// TIA Portal project "MYJZXT_PLC" (V15.1)
// 煤油加注系统(新)

(* hardware
DEVICE "S7-1200 station_1"  S7-1200 Station
   slot 0: "Rack_0"  S7-1200 Rack  Rack  V1.0
   slot 1: "PLC_1"  CPU 1215C DC/DC/Rly  6ES7 215-1HG40-0XB0  V4.2
   slot 2: "AI 8x13BIT_1"  6ES7 231-4HF32-0XB0  V2.0
   slot 3: "CB 1241 (RS485)"  CB 1241 (RS485)  6ES7 241-1CH30-1XB0  V1.0
   slot 3: "AI 8x13BIT_2"  6ES7 231-4HF32-0XB0  V2.0
   slot 4: "DI 8/DQ 8x24VDC_1"  6ES7 223-1BH32-0XB0  V2.0
*)

// ===== PLC "PLC_1"  CPU 1215C DC/DC/Rly =====

VAR_GLOBAL   // PLC tag table "默认变量表"
   "Pc0_int" AT %IW96 : Int;
   "中间变量1" AT %MD10 : Real;
   "Pc0_real" AT %MD14 : Real;
   "Pc1_int" AT %IW98 : Int;
   "Pc1_real" AT %MD18 : Real;
   "Pc2_int" AT %IW100 : Int;
   "Pc2_real" AT %MD22 : Real;
   "Pc3_int" AT %IW102 : Int;
   "Pc3_real" AT %MD26 : Real;
   "Pc4_int" AT %IW104 : Int;
   "Pc4_real" AT %MD30 : Real;
   "Pc5_int" AT %IW106 : Int;
   "Pc5_real" AT %MD34 : Real;
   "YW01_real" AT %MD38 : Real;
   "YW02_real" AT %MD42 : Real;
   "YW01_int" AT %IW112 : Int;
   "YW02_int" AT %IW114 : Int;
   "YW03_int" AT %IW116 : Int;
   "PD01" AT %IW118 : Int;
   "PD02" AT %IW120 : Int;
   "PD01_real" AT %MD50 : Real;
   "PD02_real" AT %MD54 : Real;
   "急停" AT %I0.0 : Bool;
   "变频器" AT %QW64 : Int;
   "转注泵" AT %Q0.0 : Bool;
   "加注泵" AT %Q0.1 : Bool;
   "真空泵" AT %Q0.2 : Bool;
   "DC01" AT %Q16.0 : Bool;
   "DC02" AT %Q16.1 : Bool;
   "DC03" AT %Q16.2 : Bool;
   "DC04" AT %Q16.3 : Bool;
   "DC05" AT %Q16.4 : Bool;
   "DC06" AT %Q16.5 : Bool;
   "DC07" AT %Q16.6 : Bool;
   "DC08" AT %Q16.7 : Bool;
   "变频设置" AT %MW58 : Int;
   "转注总流量" AT %MD60 : Real;
   "加注总流量" AT %MD64 : Real;
   "转注设定量" AT %MD68 : Real;
   "加注设定量" AT %MD72 : Real;
   "回排设定量" AT %MD76 : Real;
   "真空度" AT %MD6 : Real;
   "~真空加注完成" AT %M100.0 : Bool;
   "抽真空自检成功" AT %M100.1 : Bool;
   "真空加注真空自检成功" AT %M100.2 : Bool;
   "真空加注完成" AT %M100.3 : Bool;
   "回排结束标志" AT %M100.4 : Bool;
   "清洁结束" AT %M100.5 : Bool;
   "YW03_real" AT %MD46 : Real;
   "液路自检完成" AT %M100.6 : Bool;
   "转注完成" AT %M100.7 : Bool;
   "pc0" AT %MW80 : Int;
   "pc1" AT %MW82 : Int;
   "pc2" AT %MW84 : Int;
   "pc3" AT %MW86 : Int;
   "pc4" AT %MW88 : Int;
   "pc5" AT %MW90 : Int;
   "yw01" AT %MW92 : Int;
   "yw02" AT %MW94 : Int;
   "yw03" AT %MW96 : Int;
   "pd1" AT %MW98 : Int;
   "pd2" AT %MW110 : Int;
   "中间变量2" AT %MD106 : Real;
   "pip_tmp1" AT %M5.0 : Bool;
   "pip_tmp2" AT %M5.1 : Bool;
   "中间变量3" AT %MD112 : Real;
   "转/回总流量" AT %MW116 : Word;
   "加总流量" AT %MW118 : Int;
   "流量设定中间变量" AT %MW122 : Word;
   "System_Byte" AT %MB1 : Byte;
   "FirstScan" AT %M1.0 : Bool;
   "DiagStatusUpdate" AT %M1.1 : Bool;
   "AlwaysTRUE" AT %M1.2 : Bool;
   "AlwaysFALSE" AT %M1.3 : Bool;
END_VAR

VAR_GLOBAL   // PLC tag table "control"
   "current_index" AT %MB120 : Byte;   // 当前流程
   "startORstop" AT %MB124 : Byte;   // 流程开始/结束状态
   "setTime" AT %MD125 : Time;
   "current_step" AT %MB121 : Byte;
   "setZKD" AT %MW130 : Int;
   "setZKD_1" AT %MW132 : Int;
   "ZKD_keep" AT %MD134 : Real;
   "转注_set" AT %MW138 : UInt;
END_VAR

DATA_BLOCK "zhuanzhu_flow"   // DB7
{ S7_Optimized_Access := 'TRUE' }
VERSION : 0.1
// stored: InstanceOfName Flowcalc
"Flowcalc"
BEGIN
END_DATA_BLOCK

DATA_BLOCK "jiazhu_flow"   // DB8
{ S7_Optimized_Access := 'TRUE' }
VERSION : 0.1
// stored: InstanceOfName Flowcalc
"Flowcalc"
BEGIN
END_DATA_BLOCK

DATA_BLOCK "tcp_DB"   // DB9
{ S7_Optimized_Access := 'FALSE' }
VERSION : 0.1
   VAR
      ToClientArray : Array[0..50] of Byte;
      FromClientArray : Array[0..20] of Byte;
   END_VAR
BEGIN
END_DATA_BLOCK

DATA_BLOCK "tcp_status"   // DB13
{ S7_Optimized_Access := 'TRUE' }
VERSION : 0.1
   VAR
      TRCV_DONE : Bool;
      TRCV_BUSY : Bool;
      TRCV_ERROR : Bool;
      TRCV_STATUS : Word;
      TRCV_LEGNTH : UDInt;
      TSEND_DONE : Bool;
      TSEND_STATUS : Word;
      TSEND_BUSY : Bool;
      TSEND_REQ : Bool := true;
      TSEND_ERROR : Bool;
   END_VAR
BEGIN
END_DATA_BLOCK

DATA_BLOCK "485_db"   // DB30
{ S7_Optimized_Access := 'TRUE' }
VERSION : 0.1
   VAR
      "485_data" : Array[0..7] of Byte;
   END_VAR
BEGIN
END_DATA_BLOCK

// folder: System blocks/Program resources

DATA_BLOCK "timer_ylzj"   // DB1
{ S7_Optimized_Access := 'TRUE' }
AUTHOR : Simatic
FAMILY : IEC
NAME : IEC_TMR
VERSION : 1.0
// stored: InstanceOfName IEC_TIMER
"IEC_TIMER"
BEGIN
END_DATA_BLOCK

DATA_BLOCK "timer_czkzj"   // DB2
{ S7_Optimized_Access := 'TRUE' }
AUTHOR : Simatic
FAMILY : IEC
NAME : IEC_TMR
VERSION : 1.0
// stored: InstanceOfName IEC_TIMER
"IEC_TIMER"
BEGIN
END_DATA_BLOCK

DATA_BLOCK "timer_ZKD_keep"   // DB3
{ S7_Optimized_Access := 'TRUE' }
AUTHOR : Simatic
FAMILY : IEC
NAME : IEC_TMR
VERSION : 1.0
// stored: InstanceOfName IEC_TIMER
"IEC_TIMER"
BEGIN
END_DATA_BLOCK

DATA_BLOCK "timer_cqsj"   // DB4
{ S7_Optimized_Access := 'TRUE' }
AUTHOR : Simatic
FAMILY : IEC
NAME : IEC_TMR
VERSION : 1.0
// stored: InstanceOfName IEC_TIMER
"IEC_TIMER"
BEGIN
END_DATA_BLOCK

DATA_BLOCK "timer_cz"   // DB5
{ S7_Optimized_Access := 'TRUE' }
AUTHOR : Simatic
FAMILY : IEC
NAME : IEC_TMR
VERSION : 1.0
// stored: InstanceOfName IEC_TIMER
"IEC_TIMER"
BEGIN
END_DATA_BLOCK

DATA_BLOCK "timer_keeper"   // DB6
{ S7_Optimized_Access := 'TRUE' }
AUTHOR : Simatic
FAMILY : IEC
NAME : IEC_TMR
VERSION : 1.0
// stored: InstanceOfName IEC_TIMER
"IEC_TIMER"
BEGIN
END_DATA_BLOCK

DATA_BLOCK "PLC_1_Receive_DB"   // DB12
{ S7_Optimized_Access := 'TRUE' }
AUTHOR : SIMATIC
FAMILY : MC7Plus
NAME : TC_IP_v4
VERSION : 1.0
// stored: InstanceOfName TCON_IP_v4
"TCON_IP_v4"
BEGIN
   ID := 1;
   InterfaceId := 64;
   LocalPort := 2000;
   RemoteAddress.ADDR[1] := 192;
   RemoteAddress.ADDR[2] := 168;
   RemoteAddress.ADDR[3] := 2;
   RemoteAddress.ADDR[4] := 3;
END_DATA_BLOCK

DATA_BLOCK "timer_delay2"   // DB16
{ S7_Optimized_Access := 'TRUE' }
AUTHOR : Simatic
FAMILY : IEC
NAME : IEC_TMR
VERSION : 1.0
// stored: InstanceOfName IEC_TIMER
"IEC_TIMER"
BEGIN
END_DATA_BLOCK

DATA_BLOCK "IEC_Timer_0_DB_1"   // DB17
{ S7_Optimized_Access := 'TRUE' }
AUTHOR : Simatic
FAMILY : IEC
NAME : IEC_TMR
VERSION : 1.0
// stored: InstanceOfName IEC_TIMER
"IEC_TIMER"
BEGIN
END_DATA_BLOCK

DATA_BLOCK "send_delay"   // DB26
{ S7_Optimized_Access := 'TRUE' }
AUTHOR : Simatic
FAMILY : IEC
NAME : IEC_TMR
VERSION : 1.0
// stored: InstanceOfName IEC_TIMER
"IEC_TIMER"
BEGIN
END_DATA_BLOCK

DATA_BLOCK "send_delay1"   // DB27
{ S7_Optimized_Access := 'TRUE' }
AUTHOR : Simatic
FAMILY : IEC
NAME : IEC_TMR
VERSION : 1.0
// stored: InstanceOfName IEC_TIMER
"IEC_TIMER"
BEGIN
END_DATA_BLOCK

// folder: (top level)

FUNCTION_BLOCK "Flowcalc"   // FB1, SCL
{ S7_Optimized_Access := 'TRUE' }
VERSION : 0.1
   VAR_INPUT
      flow : Real;
      Enable : Bool;
   END_VAR
   VAR_OUTPUT
      sum : Real;
   END_VAR
   VAR
      data : Real;
   END_VAR
BEGIN
   IF #Enable = FALSE THEN
       #data := 0.0;
       ;
   ELSE
       IF #flow > 1.0 THEN
           #data := #data + #flow / 60 * 0.1;
           #sum := #data;
       ELSE
           #sum := #data;
       END_IF;
       // Statement section IF
       ;
   END_IF;
END_FUNCTION_BLOCK

FUNCTION "模拟量采集" : Void   // FC1, LAD
{ S7_Optimized_Access := 'TRUE' }
VERSION : 0.1
BEGIN

REGION Network 1
   // 压力传感器0
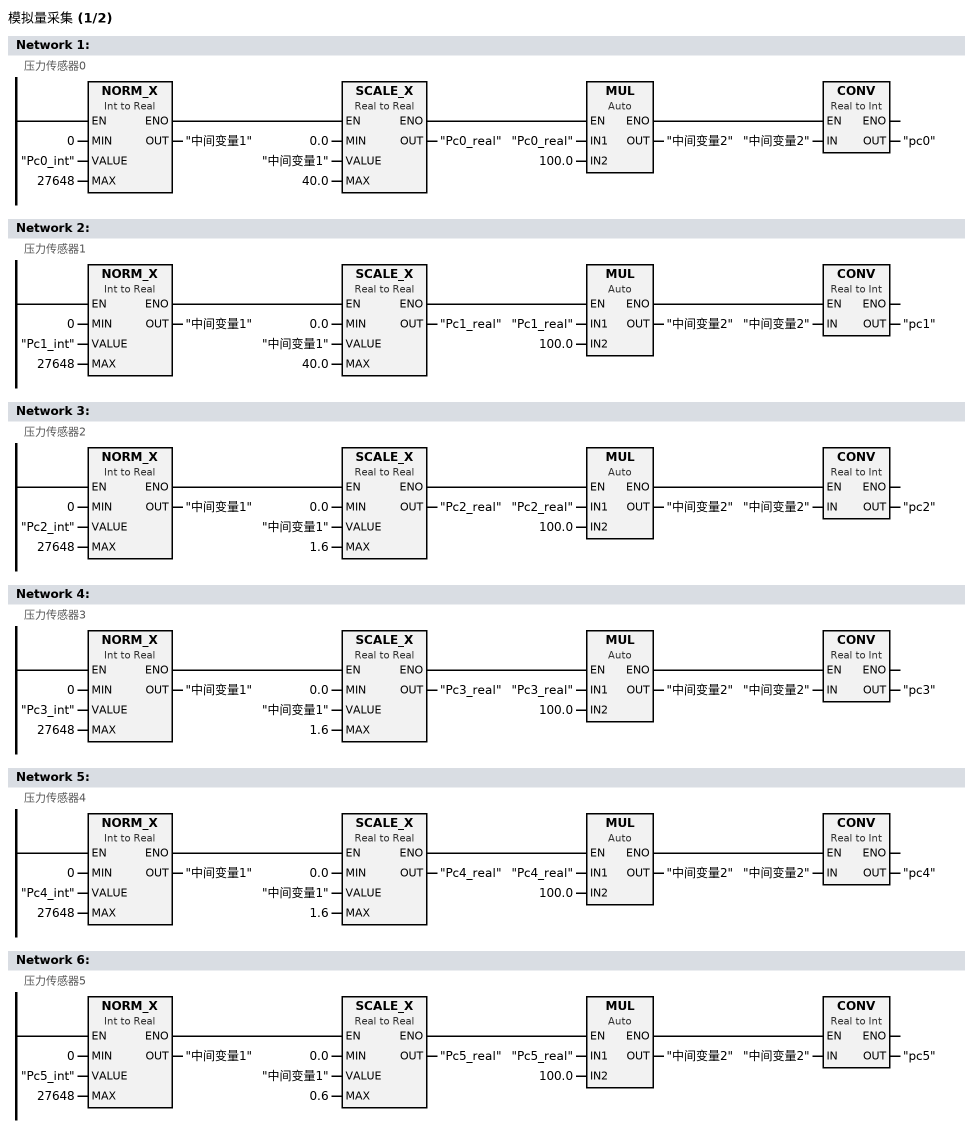
   RUNG wire#powerrail
      { S7_Templates := "[SrcType := Int, DestType := Real]"; S7_GenerateENO := "TRUE" } Normalize(min := 0, value := "Pc0_int", max := 27648, out => "中间变量1")
      { S7_Templates := "[SrcType := Real, DestType := Real]"; S7_GenerateENO := "TRUE" } Scale(min := 0.0, value := "中间变量1", max := 40.0, out => "Pc0_real")
      { S7_GenerateENO := "TRUE" } Mul(in1 := "Pc0_real", in2 := 100.0, out => "中间变量2")
      { S7_Templates := "[SrcType := Real, DestType := Int]"; S7_GenerateENO := "TRUE" } Convert(in := "中间变量2", out => "pc0")
   END_RUNG
   // the same network as SCL:
   // ENO of a box is taken as its EN; it also drops when the box reports an error
   "中间变量1" := NORM_X(MIN := 0, VALUE := "Pc0_int", MAX := 27648);
   "Pc0_real" := SCALE_X(MIN := 0.0, VALUE := "中间变量1", MAX := 40.0);
   "中间变量2" := "Pc0_real" * 100.0;
   "pc0" := REAL_TO_INT("中间变量2");
END_REGION

REGION Network 2
   // 压力传感器1
   RUNG wire#powerrail
      { S7_Templates := "[SrcType := Int, DestType := Real]"; S7_GenerateENO := "TRUE" } Normalize(min := 0, value := "Pc1_int", max := 27648, out => "中间变量1")
      { S7_Templates := "[SrcType := Real, DestType := Real]"; S7_GenerateENO := "TRUE" } Scale(min := 0.0, value := "中间变量1", max := 40.0, out => "Pc1_real")
      { S7_GenerateENO := "TRUE" } Mul(in1 := "Pc1_real", in2 := 100.0, out => "中间变量2")
      { S7_Templates := "[SrcType := Real, DestType := Int]"; S7_GenerateENO := "TRUE" } Convert(in := "中间变量2", out => "pc1")
   END_RUNG
   // the same network as SCL:
   // ENO of a box is taken as its EN; it also drops when the box reports an error
   "中间变量1" := NORM_X(MIN := 0, VALUE := "Pc1_int", MAX := 27648);
   "Pc1_real" := SCALE_X(MIN := 0.0, VALUE := "中间变量1", MAX := 40.0);
   "中间变量2" := "Pc1_real" * 100.0;
   "pc1" := REAL_TO_INT("中间变量2");
END_REGION

REGION Network 3
   // 压力传感器2
   RUNG wire#powerrail
      { S7_Templates := "[SrcType := Int, DestType := Real]"; S7_GenerateENO := "TRUE" } Normalize(min := 0, value := "Pc2_int", max := 27648, out => "中间变量1")
      { S7_Templates := "[SrcType := Real, DestType := Real]"; S7_GenerateENO := "TRUE" } Scale(min := 0.0, value := "中间变量1", max := 1.6, out => "Pc2_real")
      { S7_GenerateENO := "TRUE" } Mul(in1 := "Pc2_real", in2 := 100.0, out => "中间变量2")
      { S7_Templates := "[SrcType := Real, DestType := Int]"; S7_GenerateENO := "TRUE" } Convert(in := "中间变量2", out => "pc2")
   END_RUNG
   // the same network as SCL:
   // ENO of a box is taken as its EN; it also drops when the box reports an error
   "中间变量1" := NORM_X(MIN := 0, VALUE := "Pc2_int", MAX := 27648);
   "Pc2_real" := SCALE_X(MIN := 0.0, VALUE := "中间变量1", MAX := 1.6);
   "中间变量2" := "Pc2_real" * 100.0;
   "pc2" := REAL_TO_INT("中间变量2");
END_REGION

REGION Network 4
   // 压力传感器3
   RUNG wire#powerrail
      { S7_Templates := "[SrcType := Int, DestType := Real]"; S7_GenerateENO := "TRUE" } Normalize(min := 0, value := "Pc3_int", max := 27648, out => "中间变量1")
      { S7_Templates := "[SrcType := Real, DestType := Real]"; S7_GenerateENO := "TRUE" } Scale(min := 0.0, value := "中间变量1", max := 1.6, out => "Pc3_real")
      { S7_GenerateENO := "TRUE" } Mul(in1 := "Pc3_real", in2 := 100.0, out => "中间变量2")
      { S7_Templates := "[SrcType := Real, DestType := Int]"; S7_GenerateENO := "TRUE" } Convert(in := "中间变量2", out => "pc3")
   END_RUNG
   // the same network as SCL:
   // ENO of a box is taken as its EN; it also drops when the box reports an error
   "中间变量1" := NORM_X(MIN := 0, VALUE := "Pc3_int", MAX := 27648);
   "Pc3_real" := SCALE_X(MIN := 0.0, VALUE := "中间变量1", MAX := 1.6);
   "中间变量2" := "Pc3_real" * 100.0;
   "pc3" := REAL_TO_INT("中间变量2");
END_REGION

REGION Network 5
   // 压力传感器4
   RUNG wire#powerrail
      { S7_Templates := "[SrcType := Int, DestType := Real]"; S7_GenerateENO := "TRUE" } Normalize(min := 0, value := "Pc4_int", max := 27648, out => "中间变量1")
      { S7_Templates := "[SrcType := Real, DestType := Real]"; S7_GenerateENO := "TRUE" } Scale(min := 0.0, value := "中间变量1", max := 1.6, out => "Pc4_real")
      { S7_GenerateENO := "TRUE" } Mul(in1 := "Pc4_real", in2 := 100.0, out => "中间变量2")
      { S7_Templates := "[SrcType := Real, DestType := Int]"; S7_GenerateENO := "TRUE" } Convert(in := "中间变量2", out => "pc4")
   END_RUNG
   // the same network as SCL:
   // ENO of a box is taken as its EN; it also drops when the box reports an error
   "中间变量1" := NORM_X(MIN := 0, VALUE := "Pc4_int", MAX := 27648);
   "Pc4_real" := SCALE_X(MIN := 0.0, VALUE := "中间变量1", MAX := 1.6);
   "中间变量2" := "Pc4_real" * 100.0;
   "pc4" := REAL_TO_INT("中间变量2");
END_REGION

REGION Network 6
   // 压力传感器5
   RUNG wire#powerrail
      { S7_Templates := "[SrcType := Int, DestType := Real]"; S7_GenerateENO := "TRUE" } Normalize(min := 0, value := "Pc5_int", max := 27648, out => "中间变量1")
      { S7_Templates := "[SrcType := Real, DestType := Real]"; S7_GenerateENO := "TRUE" } Scale(min := 0.0, value := "中间变量1", max := 0.6, out => "Pc5_real")
      { S7_GenerateENO := "TRUE" } Mul(in1 := "Pc5_real", in2 := 100.0, out => "中间变量2")
      { S7_Templates := "[SrcType := Real, DestType := Int]"; S7_GenerateENO := "TRUE" } Convert(in := "中间变量2", out => "pc5")
   END_RUNG
   // the same network as SCL:
   // ENO of a box is taken as its EN; it also drops when the box reports an error
   "中间变量1" := NORM_X(MIN := 0, VALUE := "Pc5_int", MAX := 27648);
   "Pc5_real" := SCALE_X(MIN := 0.0, VALUE := "中间变量1", MAX := 0.6);
   "中间变量2" := "Pc5_real" * 100.0;
   "pc5" := REAL_TO_INT("中间变量2");
END_REGION

REGION Network 7
   // 液位计yw01
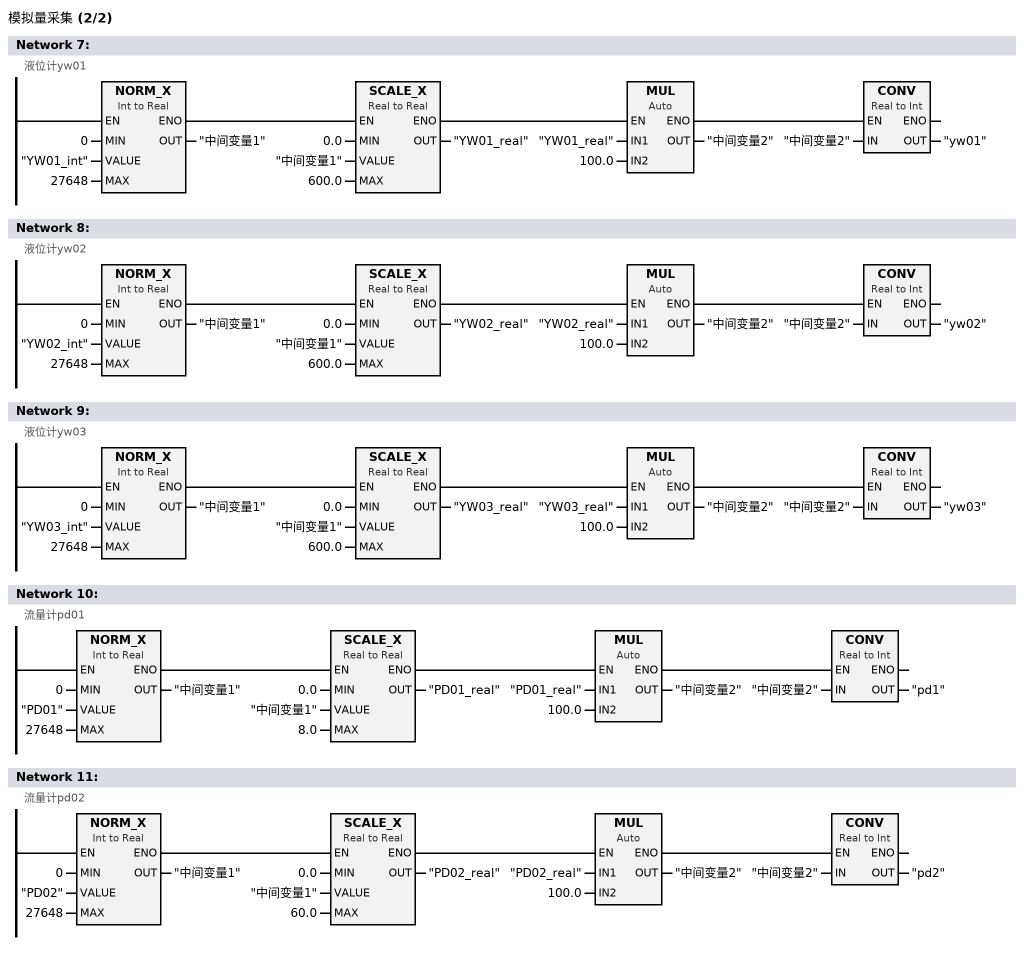
   RUNG wire#powerrail
      { S7_Templates := "[SrcType := Int, DestType := Real]"; S7_GenerateENO := "TRUE" } Normalize(min := 0, value := "YW01_int", max := 27648, out => "中间变量1")
      { S7_Templates := "[SrcType := Real, DestType := Real]"; S7_GenerateENO := "TRUE" } Scale(min := 0.0, value := "中间变量1", max := 600.0, out => "YW01_real")
      { S7_GenerateENO := "TRUE" } Mul(in1 := "YW01_real", in2 := 100.0, out => "中间变量2")
      { S7_Templates := "[SrcType := Real, DestType := Int]"; S7_GenerateENO := "TRUE" } Convert(in := "中间变量2", out => "yw01")
   END_RUNG
   // the same network as SCL:
   // ENO of a box is taken as its EN; it also drops when the box reports an error
   "中间变量1" := NORM_X(MIN := 0, VALUE := "YW01_int", MAX := 27648);
   "YW01_real" := SCALE_X(MIN := 0.0, VALUE := "中间变量1", MAX := 600.0);
   "中间变量2" := "YW01_real" * 100.0;
   "yw01" := REAL_TO_INT("中间变量2");
END_REGION

REGION Network 8
   // 液位计yw02
   RUNG wire#powerrail
      { S7_Templates := "[SrcType := Int, DestType := Real]"; S7_GenerateENO := "TRUE" } Normalize(min := 0, value := "YW02_int", max := 27648, out => "中间变量1")
      { S7_Templates := "[SrcType := Real, DestType := Real]"; S7_GenerateENO := "TRUE" } Scale(min := 0.0, value := "中间变量1", max := 600.0, out => "YW02_real")
      { S7_GenerateENO := "TRUE" } Mul(in1 := "YW02_real", in2 := 100.0, out => "中间变量2")
      { S7_Templates := "[SrcType := Real, DestType := Int]"; S7_GenerateENO := "TRUE" } Convert(in := "中间变量2", out => "yw02")
   END_RUNG
   // the same network as SCL:
   // ENO of a box is taken as its EN; it also drops when the box reports an error
   "中间变量1" := NORM_X(MIN := 0, VALUE := "YW02_int", MAX := 27648);
   "YW02_real" := SCALE_X(MIN := 0.0, VALUE := "中间变量1", MAX := 600.0);
   "中间变量2" := "YW02_real" * 100.0;
   "yw02" := REAL_TO_INT("中间变量2");
END_REGION

REGION Network 9
   // 液位计yw03
   RUNG wire#powerrail
      { S7_Templates := "[SrcType := Int, DestType := Real]"; S7_GenerateENO := "TRUE" } Normalize(min := 0, value := "YW03_int", max := 27648, out => "中间变量1")
      { S7_Templates := "[SrcType := Real, DestType := Real]"; S7_GenerateENO := "TRUE" } Scale(min := 0.0, value := "中间变量1", max := 600.0, out => "YW03_real")
      { S7_GenerateENO := "TRUE" } Mul(in1 := "YW03_real", in2 := 100.0, out => "中间变量2")
      { S7_Templates := "[SrcType := Real, DestType := Int]"; S7_GenerateENO := "TRUE" } Convert(in := "中间变量2", out => "yw03")
   END_RUNG
   // the same network as SCL:
   // ENO of a box is taken as its EN; it also drops when the box reports an error
   "中间变量1" := NORM_X(MIN := 0, VALUE := "YW03_int", MAX := 27648);
   "YW03_real" := SCALE_X(MIN := 0.0, VALUE := "中间变量1", MAX := 600.0);
   "中间变量2" := "YW03_real" * 100.0;
   "yw03" := REAL_TO_INT("中间变量2");
END_REGION

REGION Network 10
   // 流量计pd01
   RUNG wire#powerrail
      { S7_Templates := "[SrcType := Int, DestType := Real]"; S7_GenerateENO := "TRUE" } Normalize(min := 0, value := "PD01", max := 27648, out => "中间变量1")
      { S7_Templates := "[SrcType := Real, DestType := Real]"; S7_GenerateENO := "TRUE" } Scale(min := 0.0, value := "中间变量1", max := 8.0, out => "PD01_real")
      { S7_GenerateENO := "TRUE" } Mul(in1 := "PD01_real", in2 := 100.0, out => "中间变量2")
      { S7_Templates := "[SrcType := Real, DestType := Int]"; S7_GenerateENO := "TRUE" } Convert(in := "中间变量2", out => "pd1")
   END_RUNG
   // the same network as SCL:
   // ENO of a box is taken as its EN; it also drops when the box reports an error
   "中间变量1" := NORM_X(MIN := 0, VALUE := "PD01", MAX := 27648);
   "PD01_real" := SCALE_X(MIN := 0.0, VALUE := "中间变量1", MAX := 8.0);
   "中间变量2" := "PD01_real" * 100.0;
   "pd1" := REAL_TO_INT("中间变量2");
END_REGION

REGION Network 11
   // 流量计pd02
   RUNG wire#powerrail
      { S7_Templates := "[SrcType := Int, DestType := Real]"; S7_GenerateENO := "TRUE" } Normalize(min := 0, value := "PD02", max := 27648, out => "中间变量1")
      { S7_Templates := "[SrcType := Real, DestType := Real]"; S7_GenerateENO := "TRUE" } Scale(min := 0.0, value := "中间变量1", max := 60.0, out => "PD02_real")
      { S7_GenerateENO := "TRUE" } Mul(in1 := "PD02_real", in2 := 100.0, out => "中间变量2")
      { S7_Templates := "[SrcType := Real, DestType := Int]"; S7_GenerateENO := "TRUE" } Convert(in := "中间变量2", out => "pd2")
   END_RUNG
   // the same network as SCL:
   // ENO of a box is taken as its EN; it also drops when the box reports an error
   "中间变量1" := NORM_X(MIN := 0, VALUE := "PD02", MAX := 27648);
   "PD02_real" := SCALE_X(MIN := 0.0, VALUE := "中间变量1", MAX := 60.0);
   "中间变量2" := "PD02_real" * 100.0;
   "pd2" := REAL_TO_INT("中间变量2");
END_REGION
END_FUNCTION

FUNCTION "气路自检" : Void   // FC2, LAD
{ S7_Optimized_Access := 'TRUE' }
VERSION : 0.1
BEGIN

REGION Network 1: /气路自检为手动控制,当前无设置流程
END_REGION
END_FUNCTION

FUNCTION "液路自检" : Void   // FC3, LAD
{ S7_Optimized_Access := 'TRUE' }
VERSION : 0.1
   VAR_TEMP   // added for the SCL form of the ladder/FBD networks
      _w1 : Bool;
   END_VAR
BEGIN

REGION Network 1
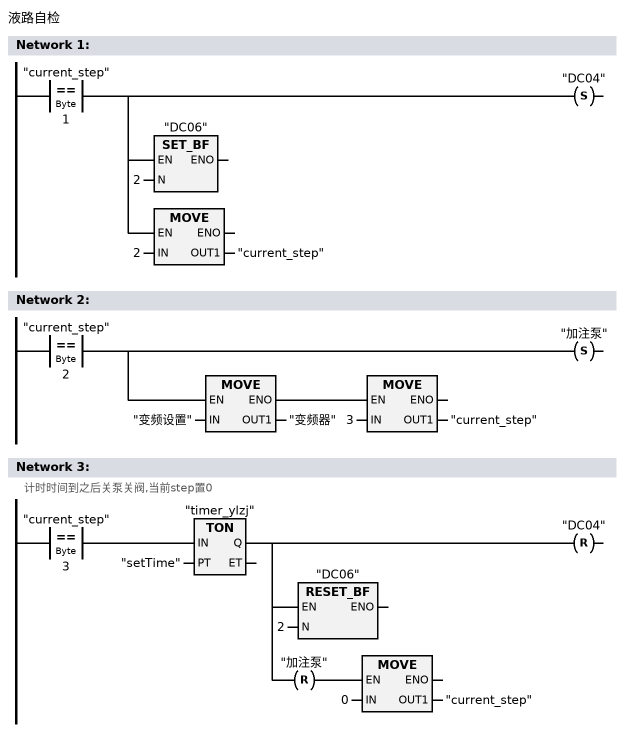
   // no SCL statement known for SBitfield: written as a call
   IF "current_step" = 1 THEN "DC04" := TRUE; END_IF;
   #_w1 := "current_step" = 1;
   IF #_w1 THEN
       SET_BF(operand := "DC06", n := 2);
       "current_step" := 2;
   END_IF;
END_REGION

REGION Network 2
   RUNG wire#powerrail
      { S7_Templates := "SrcType := Byte" } EQ_Contact(in1 := "current_step", in2 := 2)
      wire#w1
      S_Coil( "加注泵" )
   END_RUNG
   RUNG wire#w1
      { S7_GenerateENO := "TRUE" } Move(in := "变频设置", out1 => "变频器")
      { S7_GenerateENO := "TRUE" } Move(in := 3, out1 => "current_step")
   END_RUNG
   // the same network as SCL:
   // ENO of a box is taken as its EN; it also drops when the box reports an error
   IF "current_step" = 2 THEN
       "加注泵" := TRUE;
       "变频器" := "变频设置";
       "current_step" := 3;
   END_IF;
END_REGION

REGION Network 3
   // 计时时间到之后关泵关阀,当前step置0
   // no SCL statement known for RBitfield: written as a call
   "timer_ylzj".TON(IN := "current_step" = 3, PT := "setTime");
   IF "timer_ylzj".Q THEN "DC04" := FALSE; END_IF;
   #_w1 := "timer_ylzj".Q;
   IF #_w1 THEN
       RESET_BF(operand := "DC06", n := 2);
       "加注泵" := FALSE;
       "current_step" := 0;
   END_IF;
END_REGION
END_FUNCTION

FUNCTION "抽真空自检" : Void   // FC4, LAD
{ S7_Optimized_Access := 'TRUE' }
VERSION : 0.1
BEGIN

REGION Network 1
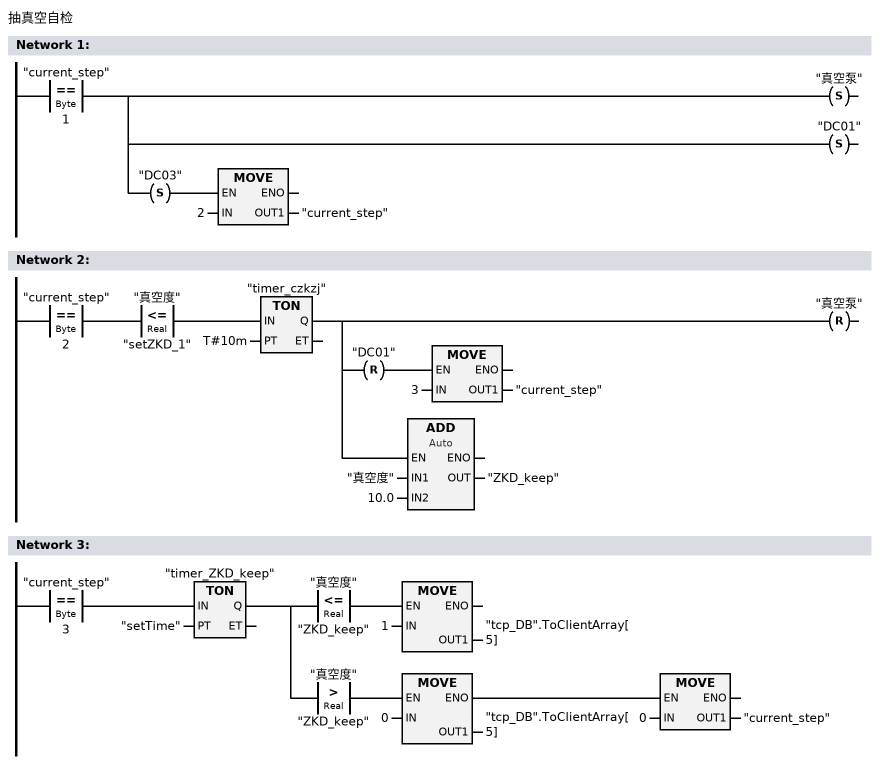
   RUNG wire#powerrail
      { S7_Templates := "SrcType := Byte" } EQ_Contact(in1 := "current_step", in2 := 1)
      wire#w1
      S_Coil( "真空泵" )
   END_RUNG
   RUNG wire#w1
      S_Coil( "DC01" )
   END_RUNG
   RUNG wire#w1
      S_Coil( "DC03" )
      { S7_GenerateENO := "TRUE" } Move(in := 2, out1 => "current_step")
   END_RUNG
   // the same network as SCL:
   IF "current_step" = 1 THEN
       "真空泵" := TRUE;
       "DC01" := TRUE;
       "DC03" := TRUE;
       "current_step" := 2;
   END_IF;
END_REGION

REGION Network 2
   "timer_czkzj".TON(IN := ("current_step" = 2) AND ("真空度" <= "setZKD_1"), PT := T#10m);
   IF "timer_czkzj".Q THEN
       "真空泵" := FALSE;
       "DC01" := FALSE;
       "current_step" := 3;
       "ZKD_keep" := "真空度" + 10.0;
   END_IF;
END_REGION

REGION Network 3
   // ENO of a box is taken as its EN; it also drops when the box reports an error
   "timer_ZKD_keep".TON(IN := "current_step" = 3, PT := "setTime");
   IF "timer_ZKD_keep".Q AND ("真空度" <= "ZKD_keep") THEN "tcp_DB".ToClientArray[5] := 1; END_IF;
   IF "timer_ZKD_keep".Q AND ("真空度" > "ZKD_keep") THEN
       "tcp_DB".ToClientArray[5] := 0;
       "current_step" := 0;
   END_IF;
END_REGION
END_FUNCTION

FUNCTION "充气流程" : Void   // FC5, LAD
{ S7_Optimized_Access := 'TRUE' }
VERSION : 0.1
   VAR_TEMP   // added for the SCL form of the ladder/FBD networks
      _w1 : Bool;
   END_VAR
BEGIN

REGION Network 1
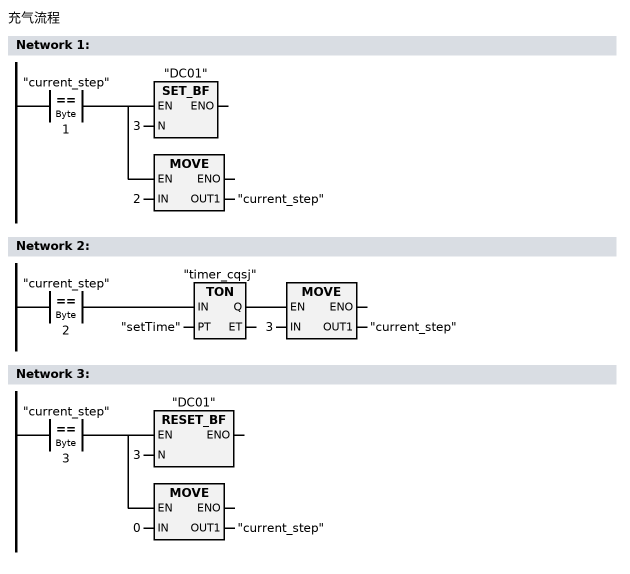
   // no SCL statement known for SBitfield: written as a call
   #_w1 := "current_step" = 1;
   IF #_w1 THEN
       SET_BF(operand := "DC01", n := 3);
       "current_step" := 2;
   END_IF;
END_REGION

REGION Network 2
   "timer_cqsj".TON(IN := "current_step" = 2, PT := "setTime");
   IF "timer_cqsj".Q THEN "current_step" := 3; END_IF;
END_REGION

REGION Network 3
   // no SCL statement known for RBitfield: written as a call
   #_w1 := "current_step" = 3;
   IF #_w1 THEN
       RESET_BF(operand := "DC01", n := 3);
       "current_step" := 0;
   END_IF;
END_REGION
END_FUNCTION

FUNCTION "抽真空急停流程" : Void   // FC6, LAD
{ S7_Optimized_Access := 'TRUE' }
VERSION : 0.1
BEGIN
END_FUNCTION

FUNCTION "煤油转注" : Void   // FC7, LAD
{ S7_Optimized_Access := 'TRUE' }
VERSION : 0.1
BEGIN

REGION Network 1
   // 开始转注打开8阀门,
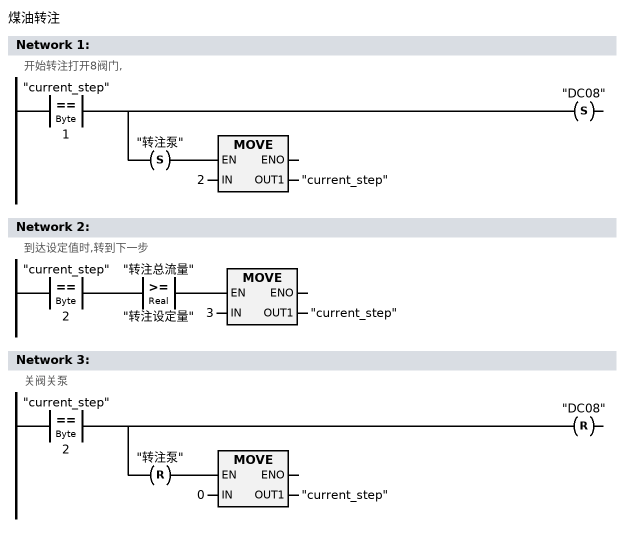
   RUNG wire#powerrail
      { S7_Templates := "SrcType := Byte" } EQ_Contact(in1 := "current_step", in2 := 1)
      wire#w1
      S_Coil( "DC08" )
   END_RUNG
   RUNG wire#w1
      S_Coil( "转注泵" )
      { S7_GenerateENO := "TRUE" } Move(in := 2, out1 => "current_step")
   END_RUNG
   // the same network as SCL:
   IF "current_step" = 1 THEN
       "DC08" := TRUE;
       "转注泵" := TRUE;
       "current_step" := 2;
   END_IF;
END_REGION

REGION Network 2
   // 到达设定值时,转到下一步
   RUNG wire#powerrail
      { S7_Templates := "SrcType := Byte" } EQ_Contact(in1 := "current_step", in2 := 2)
      { S7_Templates := "SrcType := Real" } GE_Contact(in1 := "转注总流量", in2 := "转注设定量")
      { S7_GenerateENO := "TRUE" } Move(in := 3, out1 => "current_step")
   END_RUNG
   // the same network as SCL:
   IF ("current_step" = 2) AND ("转注总流量" >= "转注设定量") THEN "current_step" := 3; END_IF;
END_REGION

REGION Network 3
   // 关阀关泵
   RUNG wire#powerrail
      { S7_Templates := "SrcType := Byte" } EQ_Contact(in1 := "current_step", in2 := 2)
      wire#w1
      R_Coil( "DC08" )
   END_RUNG
   RUNG wire#w1
      R_Coil( "转注泵" )
      { S7_GenerateENO := "TRUE" } Move(in := 0, out1 => "current_step")
   END_RUNG
   // the same network as SCL:
   IF "current_step" = 2 THEN
       "DC08" := FALSE;
       "转注泵" := FALSE;
       "current_step" := 0;
   END_IF;
END_REGION
END_FUNCTION

FUNCTION "tcp" : Void   // FC8, LAD
{ S7_Optimized_Access := 'TRUE' }
VERSION : 0.1
BEGIN

REGION Network 1
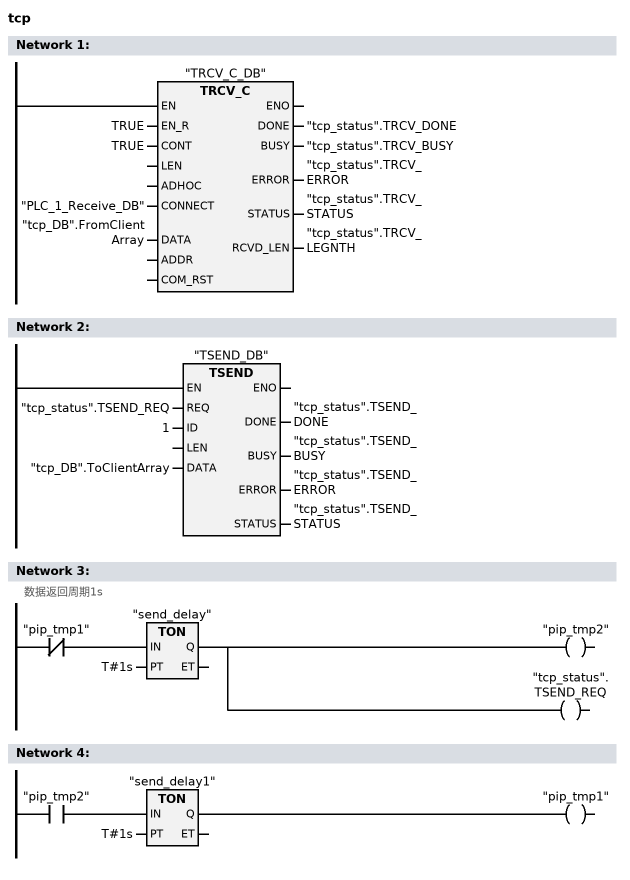
   "TRCV_C_DB"(EN_R := TRUE,   // TRCV_C
               CONT := TRUE,
               CONNECT := "PLC_1_Receive_DB",
               DATA := "tcp_DB".FromClientArray,
               DONE => "tcp_status".TRCV_DONE,
               BUSY => "tcp_status".TRCV_BUSY,
               ERROR => "tcp_status".TRCV_ERROR,
               STATUS => "tcp_status".TRCV_STATUS,
               RCVD_LEN => "tcp_status".TRCV_LEGNTH);
END_REGION

REGION Network 2
   "TSEND_DB"(REQ := "tcp_status".TSEND_REQ,   // TSEND
              ID := 1,
              DATA := "tcp_DB".ToClientArray,
              DONE => "tcp_status".TSEND_DONE,
              BUSY => "tcp_status".TSEND_BUSY,
              ERROR => "tcp_status".TSEND_ERROR,
              STATUS => "tcp_status".TSEND_STATUS);
END_REGION

REGION Network 3
   // 数据返回周期1s
   "send_delay".TON(IN := NOT "pip_tmp1", PT := T#1s);
   "pip_tmp2" := "send_delay".Q;
   "tcp_status".TSEND_REQ := "send_delay".Q;
END_REGION

REGION Network 4
   "send_delay1".TON(IN := "pip_tmp2", PT := T#1s);
   "pip_tmp1" := "send_delay1".Q;
END_REGION
END_FUNCTION

FUNCTION "Emergency" : Void   // FC9, LAD
{ S7_Optimized_Access := 'TRUE' }
VERSION : 0.1
BEGIN

REGION Network 1
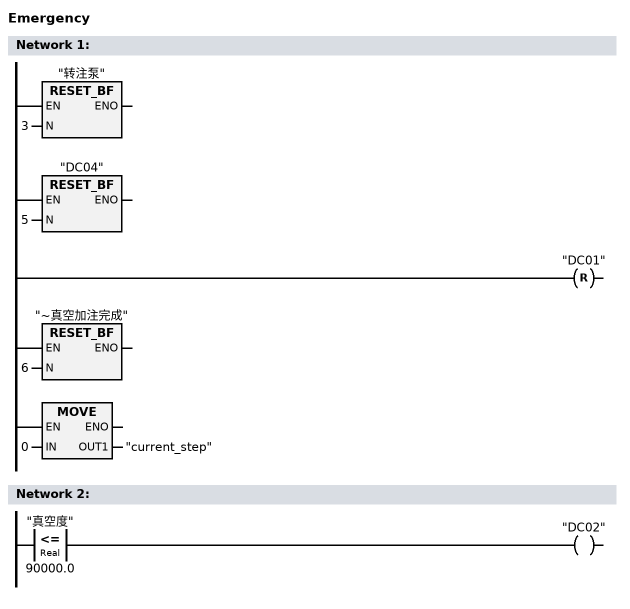
   // no SCL statement known for RBitfield: written as a call
   RESET_BF(operand := "转注泵", n := 3);
   RESET_BF(operand := "DC04", n := 5);
   "DC01" := FALSE;
   RESET_BF(operand := "~真空加注完成", n := 6);
   "current_step" := 0;
END_REGION

REGION Network 2
   RUNG wire#powerrail
      { S7_Templates := "SrcType := Real" } LE_Contact(in1 := "真空度", in2 := 90000.0)
      Coil( "DC02" )
   END_RUNG
   // the same network as SCL:
   "DC02" := "真空度" <= 90000.0;
END_REGION
END_FUNCTION

FUNCTION "煤油转注急停" : Void   // FC10, LAD
{ S7_Optimized_Access := 'TRUE' }
VERSION : 0.1
BEGIN
END_FUNCTION

FUNCTION "抽真空" : Void   // FC11, LAD
{ S7_Optimized_Access := 'TRUE' }
VERSION : 0.1
BEGIN

REGION Network 1
   // 开泵开阀
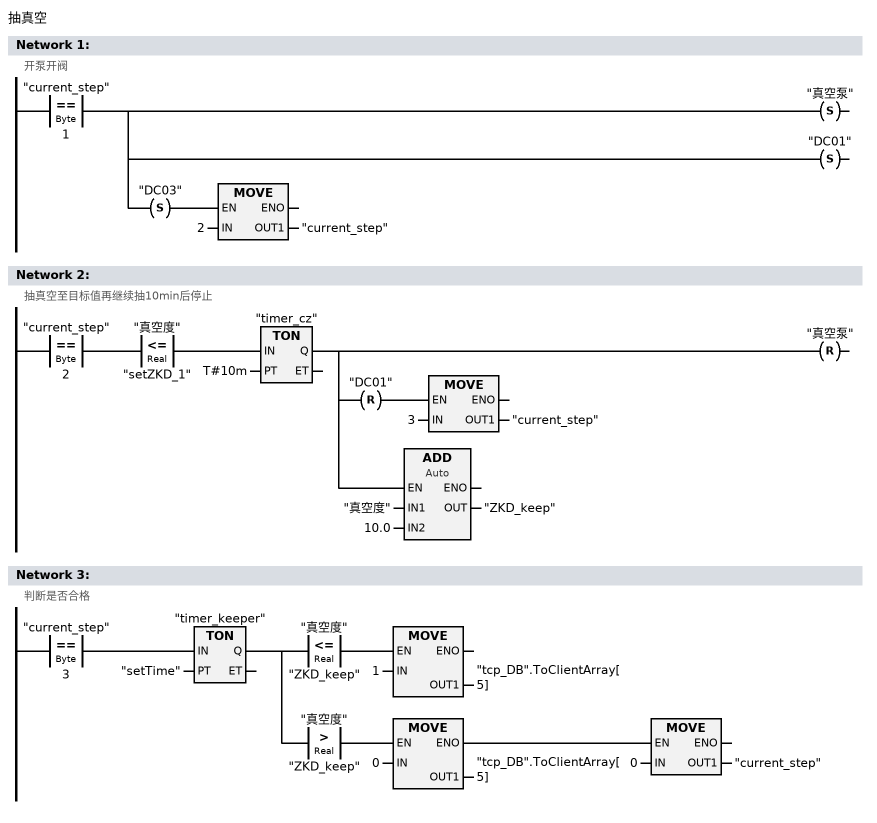
   RUNG wire#powerrail
      { S7_Templates := "SrcType := Byte" } EQ_Contact(in1 := "current_step", in2 := 1)
      wire#w1
      S_Coil( "真空泵" )
   END_RUNG
   RUNG wire#w1
      S_Coil( "DC01" )
   END_RUNG
   RUNG wire#w1
      S_Coil( "DC03" )
      { S7_GenerateENO := "TRUE" } Move(in := 2, out1 => "current_step")
   END_RUNG
   // the same network as SCL:
   IF "current_step" = 1 THEN
       "真空泵" := TRUE;
       "DC01" := TRUE;
       "DC03" := TRUE;
       "current_step" := 2;
   END_IF;
END_REGION

REGION Network 2
   // 抽真空至目标值再继续抽10min后停止
   "timer_cz".TON(IN := ("current_step" = 2) AND ("真空度" <= "setZKD_1"), PT := T#10m);
   IF "timer_cz".Q THEN
       "真空泵" := FALSE;
       "DC01" := FALSE;
       "current_step" := 3;
       "ZKD_keep" := "真空度" + 10.0;
   END_IF;
END_REGION

REGION Network 3
   // 判断是否合格
   // ENO of a box is taken as its EN; it also drops when the box reports an error
   "timer_keeper".TON(IN := "current_step" = 3, PT := "setTime");
   IF "timer_keeper".Q AND ("真空度" <= "ZKD_keep") THEN "tcp_DB".ToClientArray[5] := 1; END_IF;
   IF "timer_keeper".Q AND ("真空度" > "ZKD_keep") THEN
       "tcp_DB".ToClientArray[5] := 0;
       "current_step" := 0;
   END_IF;
END_REGION
END_FUNCTION

FUNCTION "煤油加注" : Void   // FC12, LAD
{ S7_Optimized_Access := 'TRUE' }
VERSION : 0.1
   VAR_TEMP   // added for the SCL form of the ladder/FBD networks
      _w1 : Bool;
   END_VAR
BEGIN

REGION Network 1
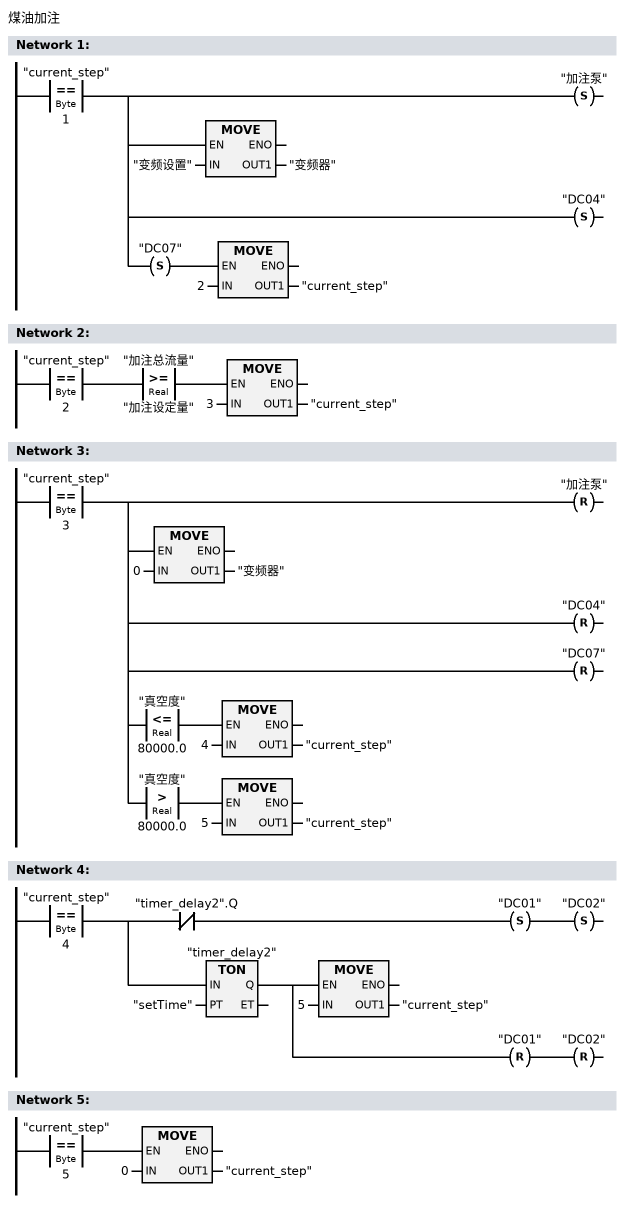
   RUNG wire#powerrail
      { S7_Templates := "SrcType := Byte" } EQ_Contact(in1 := "current_step", in2 := 1)
      wire#w1
      S_Coil( "加注泵" )
   END_RUNG
   RUNG wire#w1
      { S7_GenerateENO := "TRUE" } Move(in := "变频设置", out1 => "变频器")
   END_RUNG
   RUNG wire#w1
      S_Coil( "DC04" )
   END_RUNG
   RUNG wire#w1
      S_Coil( "DC07" )
      { S7_GenerateENO := "TRUE" } Move(in := 2, out1 => "current_step")
   END_RUNG
   // the same network as SCL:
   IF "current_step" = 1 THEN
       "加注泵" := TRUE;
       "变频器" := "变频设置";
       "DC04" := TRUE;
       "DC07" := TRUE;
       "current_step" := 2;
   END_IF;
END_REGION

REGION Network 2
   RUNG wire#powerrail
      { S7_Templates := "SrcType := Byte" } EQ_Contact(in1 := "current_step", in2 := 2)
      { S7_Templates := "SrcType := Real" } GE_Contact(in1 := "加注总流量", in2 := "加注设定量")
      { S7_GenerateENO := "TRUE" } Move(in := 3, out1 => "current_step")
   END_RUNG
   // the same network as SCL:
   IF ("current_step" = 2) AND ("加注总流量" >= "加注设定量") THEN "current_step" := 3; END_IF;
END_REGION

REGION Network 3
   RUNG wire#powerrail
      { S7_Templates := "SrcType := Byte" } EQ_Contact(in1 := "current_step", in2 := 3)
      wire#w1
      R_Coil( "加注泵" )
   END_RUNG
   RUNG wire#w1
      { S7_GenerateENO := "TRUE" } Move(in := 0, out1 => "变频器")
   END_RUNG
   RUNG wire#w1
      R_Coil( "DC04" )
   END_RUNG
   RUNG wire#w1
      R_Coil( "DC07" )
   END_RUNG
   RUNG wire#w1
      { S7_Templates := "SrcType := Real" } LE_Contact(in1 := "真空度", in2 := 80000.0)
      { S7_GenerateENO := "TRUE" } Move(in := 4, out1 => "current_step")
   END_RUNG
   RUNG wire#w1
      { S7_Templates := "SrcType := Real" } GT_Contact(in1 := "真空度", in2 := 80000.0)
      { S7_GenerateENO := "TRUE" } Move(in := 5, out1 => "current_step")
   END_RUNG
   // the same network as SCL:
   #_w1 := "current_step" = 3;
   IF #_w1 THEN
       "加注泵" := FALSE;
       "变频器" := 0;
       "DC04" := FALSE;
       "DC07" := FALSE;
   END_IF;
   IF #_w1 AND ("真空度" <= 80000.0) THEN "current_step" := 4; END_IF;
   IF #_w1 AND ("真空度" > 80000.0) THEN "current_step" := 5; END_IF;
END_REGION

REGION Network 4
   #_w1 := "current_step" = 4;
   IF #_w1 AND NOT "timer_delay2".Q THEN
       "DC01" := TRUE;
       "DC02" := TRUE;
   END_IF;
   "timer_delay2".TON(IN := #_w1, PT := "setTime");
   IF "timer_delay2".Q THEN
       "current_step" := 5;
       "DC01" := FALSE;
       "DC02" := FALSE;
   END_IF;
END_REGION

REGION Network 5
   RUNG wire#powerrail
      { S7_Templates := "SrcType := Byte" } EQ_Contact(in1 := "current_step", in2 := 5)
      { S7_GenerateENO := "TRUE" } Move(in := 0, out1 => "current_step")
   END_RUNG
   // the same network as SCL:
   IF "current_step" = 5 THEN "current_step" := 0; END_IF;
END_REGION
END_FUNCTION

FUNCTION "modbus" : Void   // FC13, LAD
{ S7_Optimized_Access := 'TRUE' }
VERSION : 0.1
BEGIN

REGION Network 1
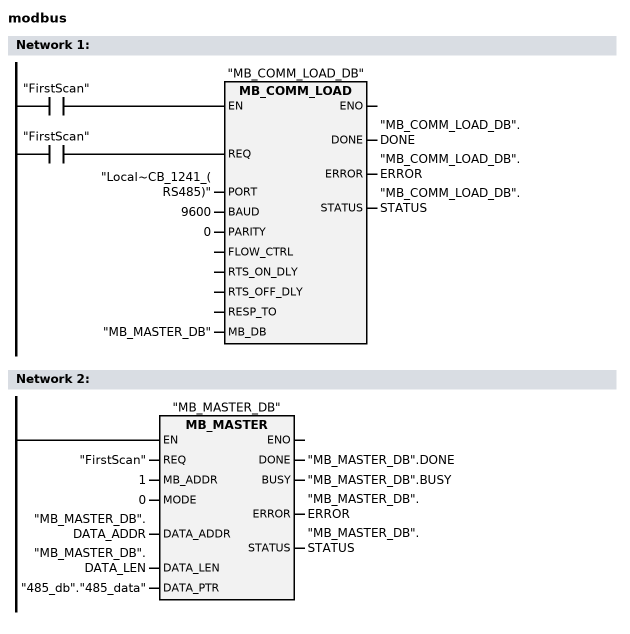
   IF "FirstScan" THEN
       "MB_COMM_LOAD_DB"(REQ := "FirstScan",   // MB_COMM_LOAD
                         PORT := "Local~CB_1241_(RS485)",
                         BAUD := 9600,
                         PARITY := 0,
                         MB_DB := "MB_MASTER_DB",
                         DONE => "MB_COMM_LOAD_DB".DONE,
                         ERROR => "MB_COMM_LOAD_DB".ERROR,
                         STATUS => "MB_COMM_LOAD_DB".STATUS);
   END_IF;
END_REGION

REGION Network 2
   "MB_MASTER_DB"(REQ := "FirstScan",   // MB_MASTER
                  MB_ADDR := 1,
                  MODE := 0,
                  DATA_ADDR := "MB_MASTER_DB".DATA_ADDR,
                  DATA_LEN := "MB_MASTER_DB".DATA_LEN,
                  DATA_PTR := "485_db"."485_data",
                  DONE => "MB_MASTER_DB".DONE,
                  BUSY => "MB_MASTER_DB".BUSY,
                  ERROR => "MB_MASTER_DB".ERROR,
                  STATUS => "MB_MASTER_DB".STATUS);
END_REGION
END_FUNCTION

FUNCTION "煤油加注急停" : Void   // FC14, LAD
{ S7_Optimized_Access := 'TRUE' }
VERSION : 0.1
BEGIN
END_FUNCTION

FUNCTION "煤油回排" : Void   // FC15, LAD
{ S7_Optimized_Access := 'TRUE' }
VERSION : 0.1
   VAR_TEMP   // added for the SCL form of the ladder/FBD networks
      _w1 : Bool;
   END_VAR
BEGIN

REGION Network 1
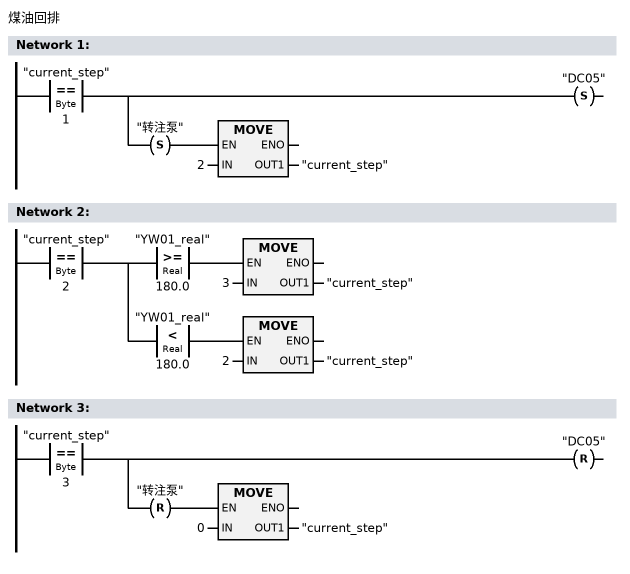
   RUNG wire#powerrail
      { S7_Templates := "SrcType := Byte" } EQ_Contact(in1 := "current_step", in2 := 1)
      wire#w1
      S_Coil( "DC05" )
   END_RUNG
   RUNG wire#w1
      S_Coil( "转注泵" )
      { S7_GenerateENO := "TRUE" } Move(in := 2, out1 => "current_step")
   END_RUNG
   // the same network as SCL:
   IF "current_step" = 1 THEN
       "DC05" := TRUE;
       "转注泵" := TRUE;
       "current_step" := 2;
   END_IF;
END_REGION

REGION Network 2
   RUNG wire#powerrail
      { S7_Templates := "SrcType := Byte" } EQ_Contact(in1 := "current_step", in2 := 2)
      wire#w1
      { S7_Templates := "SrcType := Real" } GE_Contact(in1 := "YW01_real", in2 := 180.0)
      { S7_GenerateENO := "TRUE" } Move(in := 3, out1 => "current_step")
   END_RUNG
   RUNG wire#w1
      { S7_Templates := "SrcType := Real" } LT_Contact(in1 := "YW01_real", in2 := 180.0)
      { S7_GenerateENO := "TRUE" } Move(in := 2, out1 => "current_step")
   END_RUNG
   // the same network as SCL:
   #_w1 := "current_step" = 2;
   IF #_w1 AND ("YW01_real" >= 180.0) THEN "current_step" := 3; END_IF;
   IF #_w1 AND ("YW01_real" < 180.0) THEN "current_step" := 2; END_IF;
END_REGION

REGION Network 3
   RUNG wire#powerrail
      { S7_Templates := "SrcType := Byte" } EQ_Contact(in1 := "current_step", in2 := 3)
      wire#w1
      R_Coil( "DC05" )
   END_RUNG
   RUNG wire#w1
      R_Coil( "转注泵" )
      { S7_GenerateENO := "TRUE" } Move(in := 0, out1 => "current_step")
   END_RUNG
   // the same network as SCL:
   IF "current_step" = 3 THEN
       "DC05" := FALSE;
       "转注泵" := FALSE;
       "current_step" := 0;
   END_IF;
END_REGION
END_FUNCTION

FUNCTION "煤油回排急停" : Void   // FC16, LAD
{ S7_Optimized_Access := 'TRUE' }
VERSION : 0.1
BEGIN
END_FUNCTION

FUNCTION "煤油清洁" : Void   // FC17, LAD
{ S7_Optimized_Access := 'TRUE' }
VERSION : 0.1
BEGIN

REGION Network 1
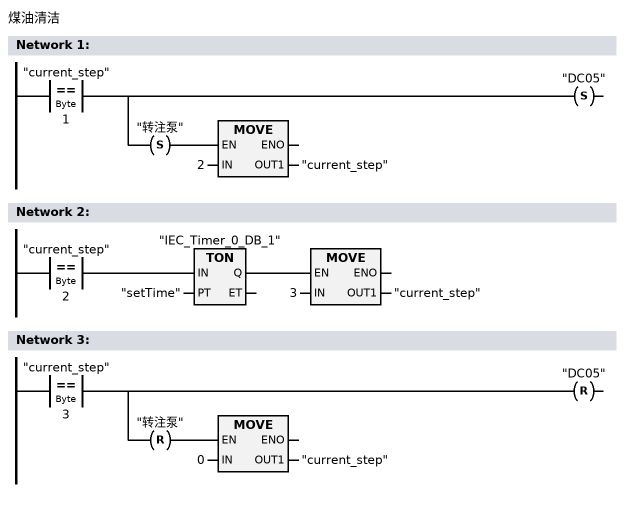
   RUNG wire#powerrail
      { S7_Templates := "SrcType := Byte" } EQ_Contact(in1 := "current_step", in2 := 1)
      wire#w1
      S_Coil( "DC05" )
   END_RUNG
   RUNG wire#w1
      S_Coil( "转注泵" )
      { S7_GenerateENO := "TRUE" } Move(in := 2, out1 => "current_step")
   END_RUNG
   // the same network as SCL:
   IF "current_step" = 1 THEN
       "DC05" := TRUE;
       "转注泵" := TRUE;
       "current_step" := 2;
   END_IF;
END_REGION

REGION Network 2
   "IEC_Timer_0_DB_1".TON(IN := "current_step" = 2, PT := "setTime");
   IF "IEC_Timer_0_DB_1".Q THEN "current_step" := 3; END_IF;
END_REGION

REGION Network 3
   RUNG wire#powerrail
      { S7_Templates := "SrcType := Byte" } EQ_Contact(in1 := "current_step", in2 := 3)
      wire#w1
      R_Coil( "DC05" )
   END_RUNG
   RUNG wire#w1
      R_Coil( "转注泵" )
      { S7_GenerateENO := "TRUE" } Move(in := 0, out1 => "current_step")
   END_RUNG
   // the same network as SCL:
   IF "current_step" = 3 THEN
       "DC05" := FALSE;
       "转注泵" := FALSE;
       "current_step" := 0;
   END_IF;
END_REGION
END_FUNCTION

FUNCTION "tcp发送数据" : Void   // FC18, LAD
{ S7_Optimized_Access := 'TRUE' }
VERSION : 0.1
BEGIN

REGION Network 1
   // tcp发送当前流程序号
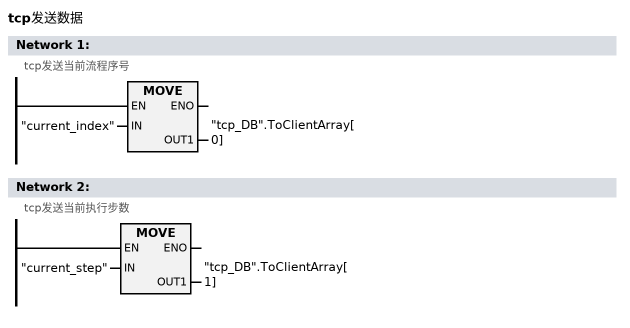
   RUNG wire#powerrail
      { S7_GenerateENO := "TRUE" } Move(in := "current_index", out1 => "tcp_DB".ToClientArray[0])
   END_RUNG
   // the same network as SCL:
   "tcp_DB".ToClientArray[0] := "current_index";
END_REGION

REGION Network 2
   // tcp发送当前执行步数
   RUNG wire#powerrail
      { S7_GenerateENO := "TRUE" } Move(in := "current_step", out1 => "tcp_DB".ToClientArray[1])
   END_RUNG
   // the same network as SCL:
   "tcp_DB".ToClientArray[1] := "current_step";
END_REGION
END_FUNCTION

FUNCTION "tcp接收数据" : Void   // FC19, LAD
{ S7_Optimized_Access := 'TRUE' }
VERSION : 0.1
BEGIN

REGION Network 1
   // 当前无流程执行时,从tcp数据byte[0]获取当前流程序号,当前执行步数置1
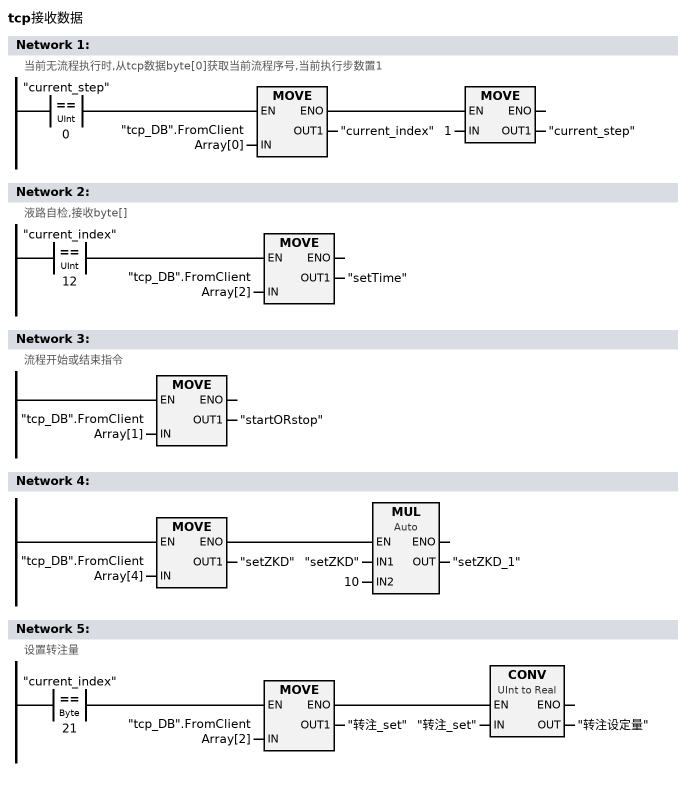
   RUNG wire#powerrail
      { S7_Templates := "SrcType := UInt" } EQ_Contact(in1 := "current_step", in2 := 0)
      { S7_GenerateENO := "TRUE" } Move(in := "tcp_DB".FromClientArray[0], out1 => "current_index")
      { S7_GenerateENO := "TRUE" } Move(in := 1, out1 => "current_step")
   END_RUNG
   // the same network as SCL:
   // ENO of a box is taken as its EN; it also drops when the box reports an error
   IF "current_step" = 0 THEN
       "current_index" := "tcp_DB".FromClientArray[0];
       "current_step" := 1;
   END_IF;
END_REGION

REGION Network 2
   // 液路自检,接收byte[]
   RUNG wire#powerrail
      { S7_Templates := "SrcType := UInt" } EQ_Contact(in1 := "current_index", in2 := 12)
      { S7_GenerateENO := "TRUE" } Move(in := "tcp_DB".FromClientArray[2], out1 => "setTime")
   END_RUNG
   // the same network as SCL:
   IF "current_index" = 12 THEN "setTime" := "tcp_DB".FromClientArray[2]; END_IF;
END_REGION

REGION Network 3
   // 流程开始或结束指令
   RUNG wire#powerrail
      { S7_GenerateENO := "TRUE" } Move(in := "tcp_DB".FromClientArray[1], out1 => "startORstop")
   END_RUNG
   // the same network as SCL:
   "startORstop" := "tcp_DB".FromClientArray[1];
END_REGION

REGION Network 4
   RUNG wire#powerrail
      { S7_GenerateENO := "TRUE" } Move(in := "tcp_DB".FromClientArray[4], out1 => "setZKD")
      { S7_GenerateENO := "TRUE" } Mul(in1 := "setZKD", in2 := 10, out => "setZKD_1")
   END_RUNG
   // the same network as SCL:
   // ENO of a box is taken as its EN; it also drops when the box reports an error
   "setZKD" := "tcp_DB".FromClientArray[4];
   "setZKD_1" := "setZKD" * 10;
END_REGION

REGION Network 5
   // 设置转注量
   RUNG wire#powerrail
      { S7_Templates := "SrcType := Byte" } EQ_Contact(in1 := "current_index", in2 := 21)
      { S7_GenerateENO := "TRUE" } Move(in := "tcp_DB".FromClientArray[2], out1 => "转注_set")
      { S7_Templates := "[SrcType := UInt, DestType := Real]"; S7_GenerateENO := "TRUE" } Convert(in := "转注_set", out => "转注设定量")
   END_RUNG
   // the same network as SCL:
   // ENO of a box is taken as its EN; it also drops when the box reports an error
   IF "current_index" = 21 THEN
       "转注_set" := "tcp_DB".FromClientArray[2];
       "转注设定量" := UINT_TO_REAL("转注_set");
   END_IF;
END_REGION
END_FUNCTION

FUNCTION "程序停止" : Void   // FC20, LAD
{ S7_Optimized_Access := 'TRUE' }
VERSION : 0.1
BEGIN

REGION Network 1
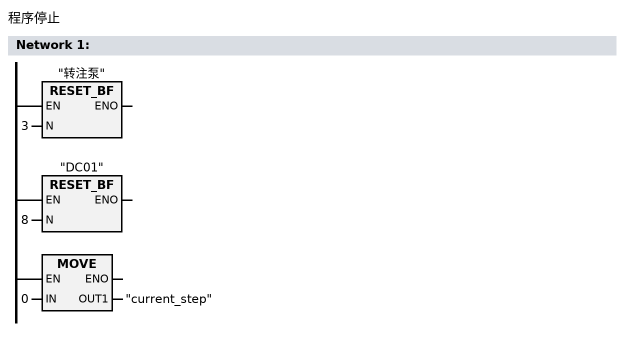
   // no SCL statement known for RBitfield: written as a call
   RESET_BF(operand := "转注泵", n := 3);
   RESET_BF(operand := "DC01", n := 8);
   "current_step" := 0;
END_REGION
END_FUNCTION

ORGANIZATION_BLOCK "Main"   // OB1, LAD, ProgramCycle
TITLE = "Main Program Sweep (Cycle)"
{ S7_Optimized_Access := 'TRUE' }
VERSION : 0.1
   VAR_INPUT
      Initial_Call : Bool;   // Initial call of this OB
      Remanence : Bool;   // =True, if remanent data are available
   END_VAR
BEGIN

REGION Network 1: 模拟量采集
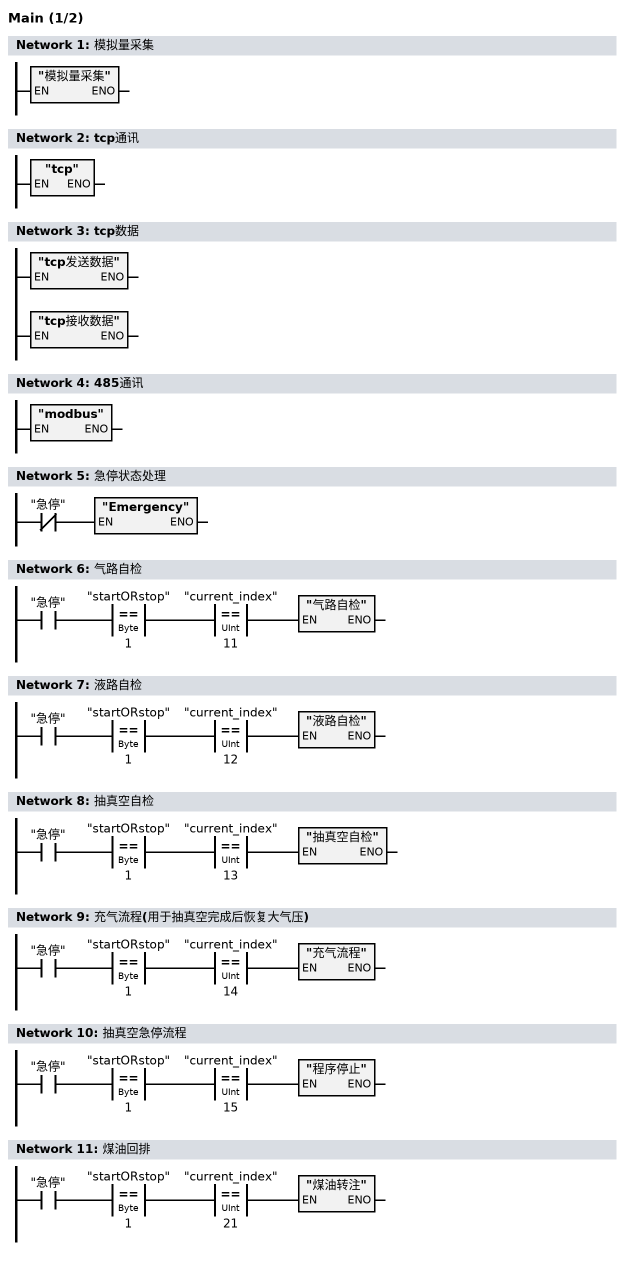
   RUNG wire#powerrail
      "模拟量采集"()
   END_RUNG
   // the same network as SCL:
   "模拟量采集"();
END_REGION

REGION Network 2: tcp通讯
   RUNG wire#powerrail
      "tcp"()
   END_RUNG
   // the same network as SCL:
   "tcp"();
END_REGION

REGION Network 3: tcp数据
   RUNG wire#powerrail
      "tcp发送数据"()
   END_RUNG
   RUNG wire#powerrail
      "tcp接收数据"()
   END_RUNG
   // the same network as SCL:
   "tcp发送数据"();
   "tcp接收数据"();
END_REGION

REGION Network 4: 485通讯
   RUNG wire#powerrail
      "modbus"()
   END_RUNG
   // the same network as SCL:
   "modbus"();
END_REGION

REGION Network 5: 急停状态处理
   RUNG wire#powerrail
      I_Contact( "急停" )
      "Emergency"()
   END_RUNG
   // the same network as SCL:
   IF NOT "急停" THEN "Emergency"(); END_IF;
END_REGION

REGION Network 6: 气路自检
   RUNG wire#powerrail
      Contact( "急停" )
      { S7_Templates := "SrcType := Byte" } EQ_Contact(in1 := "startORstop", in2 := 1)
      { S7_Templates := "SrcType := UInt" } EQ_Contact(in1 := "current_index", in2 := 11)
      "气路自检"()
   END_RUNG
   // the same network as SCL:
   IF "急停" AND ("startORstop" = 1) AND ("current_index" = 11) THEN "气路自检"(); END_IF;
END_REGION

REGION Network 7: 液路自检
   RUNG wire#powerrail
      Contact( "急停" )
      { S7_Templates := "SrcType := Byte" } EQ_Contact(in1 := "startORstop", in2 := 1)
      { S7_Templates := "SrcType := UInt" } EQ_Contact(in1 := "current_index", in2 := 12)
      "液路自检"()
   END_RUNG
   // the same network as SCL:
   IF "急停" AND ("startORstop" = 1) AND ("current_index" = 12) THEN "液路自检"(); END_IF;
END_REGION

REGION Network 8: 抽真空自检
   RUNG wire#powerrail
      Contact( "急停" )
      { S7_Templates := "SrcType := Byte" } EQ_Contact(in1 := "startORstop", in2 := 1)
      { S7_Templates := "SrcType := UInt" } EQ_Contact(in1 := "current_index", in2 := 13)
      "抽真空自检"()
   END_RUNG
   // the same network as SCL:
   IF "急停" AND ("startORstop" = 1) AND ("current_index" = 13) THEN "抽真空自检"(); END_IF;
END_REGION

REGION Network 9: 充气流程(用于抽真空完成后恢复大气压)
   RUNG wire#powerrail
      Contact( "急停" )
      { S7_Templates := "SrcType := Byte" } EQ_Contact(in1 := "startORstop", in2 := 1)
      { S7_Templates := "SrcType := UInt" } EQ_Contact(in1 := "current_index", in2 := 14)
      "充气流程"()
   END_RUNG
   // the same network as SCL:
   IF "急停" AND ("startORstop" = 1) AND ("current_index" = 14) THEN "充气流程"(); END_IF;
END_REGION

REGION Network 10: 抽真空急停流程
   RUNG wire#powerrail
      Contact( "急停" )
      { S7_Templates := "SrcType := Byte" } EQ_Contact(in1 := "startORstop", in2 := 1)
      { S7_Templates := "SrcType := UInt" } EQ_Contact(in1 := "current_index", in2 := 15)
      "程序停止"()
   END_RUNG
   // the same network as SCL:
   IF "急停" AND ("startORstop" = 1) AND ("current_index" = 15) THEN "程序停止"(); END_IF;
END_REGION

REGION Network 11: 煤油回排
   RUNG wire#powerrail
      Contact( "急停" )
      { S7_Templates := "SrcType := Byte" } EQ_Contact(in1 := "startORstop", in2 := 1)
      { S7_Templates := "SrcType := UInt" } EQ_Contact(in1 := "current_index", in2 := 21)
      "煤油转注"()
   END_RUNG
   // the same network as SCL:
   IF "急停" AND ("startORstop" = 1) AND ("current_index" = 21) THEN "煤油转注"(); END_IF;
END_REGION

REGION Network 12: 煤油转注急停
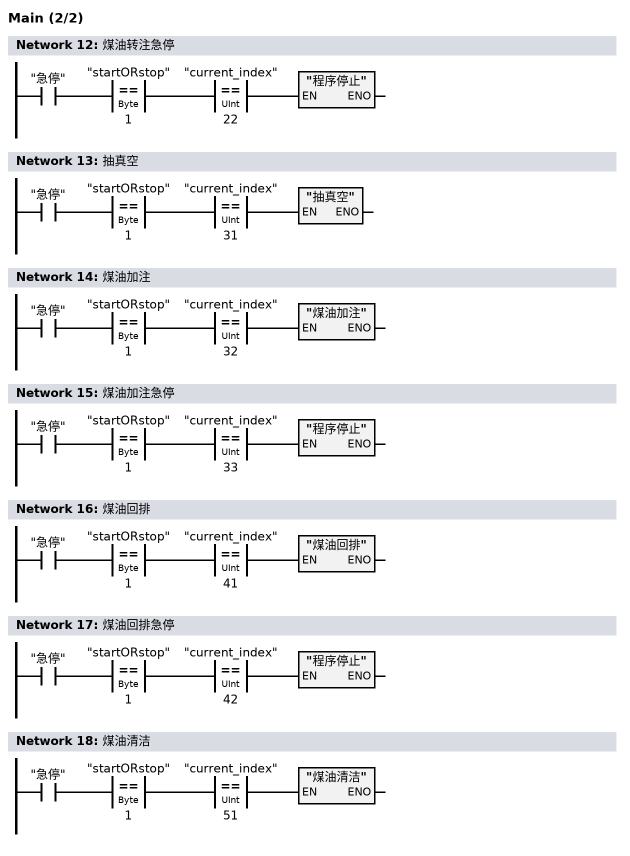
   RUNG wire#powerrail
      Contact( "急停" )
      { S7_Templates := "SrcType := Byte" } EQ_Contact(in1 := "startORstop", in2 := 1)
      { S7_Templates := "SrcType := UInt" } EQ_Contact(in1 := "current_index", in2 := 22)
      "程序停止"()
   END_RUNG
   // the same network as SCL:
   IF "急停" AND ("startORstop" = 1) AND ("current_index" = 22) THEN "程序停止"(); END_IF;
END_REGION

REGION Network 13: 抽真空
   RUNG wire#powerrail
      Contact( "急停" )
      { S7_Templates := "SrcType := Byte" } EQ_Contact(in1 := "startORstop", in2 := 1)
      { S7_Templates := "SrcType := UInt" } EQ_Contact(in1 := "current_index", in2 := 31)
      "抽真空"()
   END_RUNG
   // the same network as SCL:
   IF "急停" AND ("startORstop" = 1) AND ("current_index" = 31) THEN "抽真空"(); END_IF;
END_REGION

REGION Network 14: 煤油加注
   RUNG wire#powerrail
      Contact( "急停" )
      { S7_Templates := "SrcType := Byte" } EQ_Contact(in1 := "startORstop", in2 := 1)
      { S7_Templates := "SrcType := UInt" } EQ_Contact(in1 := "current_index", in2 := 32)
      "煤油加注"()
   END_RUNG
   // the same network as SCL:
   IF "急停" AND ("startORstop" = 1) AND ("current_index" = 32) THEN "煤油加注"(); END_IF;
END_REGION

REGION Network 15: 煤油加注急停
   RUNG wire#powerrail
      Contact( "急停" )
      { S7_Templates := "SrcType := Byte" } EQ_Contact(in1 := "startORstop", in2 := 1)
      { S7_Templates := "SrcType := UInt" } EQ_Contact(in1 := "current_index", in2 := 33)
      "程序停止"()
   END_RUNG
   // the same network as SCL:
   IF "急停" AND ("startORstop" = 1) AND ("current_index" = 33) THEN "程序停止"(); END_IF;
END_REGION

REGION Network 16: 煤油回排
   RUNG wire#powerrail
      Contact( "急停" )
      { S7_Templates := "SrcType := Byte" } EQ_Contact(in1 := "startORstop", in2 := 1)
      { S7_Templates := "SrcType := UInt" } EQ_Contact(in1 := "current_index", in2 := 41)
      "煤油回排"()
   END_RUNG
   // the same network as SCL:
   IF "急停" AND ("startORstop" = 1) AND ("current_index" = 41) THEN "煤油回排"(); END_IF;
END_REGION

REGION Network 17: 煤油回排急停
   RUNG wire#powerrail
      Contact( "急停" )
      { S7_Templates := "SrcType := Byte" } EQ_Contact(in1 := "startORstop", in2 := 1)
      { S7_Templates := "SrcType := UInt" } EQ_Contact(in1 := "current_index", in2 := 42)
      "程序停止"()
   END_RUNG
   // the same network as SCL:
   IF "急停" AND ("startORstop" = 1) AND ("current_index" = 42) THEN "程序停止"(); END_IF;
END_REGION

REGION Network 18: 煤油清洁
   RUNG wire#powerrail
      Contact( "急停" )
      { S7_Templates := "SrcType := Byte" } EQ_Contact(in1 := "startORstop", in2 := 1)
      { S7_Templates := "SrcType := UInt" } EQ_Contact(in1 := "current_index", in2 := 51)
      "煤油清洁"()
   END_RUNG
   // the same network as SCL:
   IF "急停" AND ("startORstop" = 1) AND ("current_index" = 51) THEN "煤油清洁"(); END_IF;
END_REGION
END_ORGANIZATION_BLOCK

ORGANIZATION_BLOCK "Cyclic interrupt"   // OB30, LAD, CyclicInterrupt
{ S7_Optimized_Access := 'TRUE' }
VERSION : 0.1
   VAR_INPUT
      Initial_Call : Bool;   // Initial call of this OB
      Event_Count : Int;   // Events discarded
   END_VAR
   VAR_TEMP   // added for the SCL form of the ladder/FBD networks
      _w1 : Bool;
   END_VAR
BEGIN

REGION Network 1
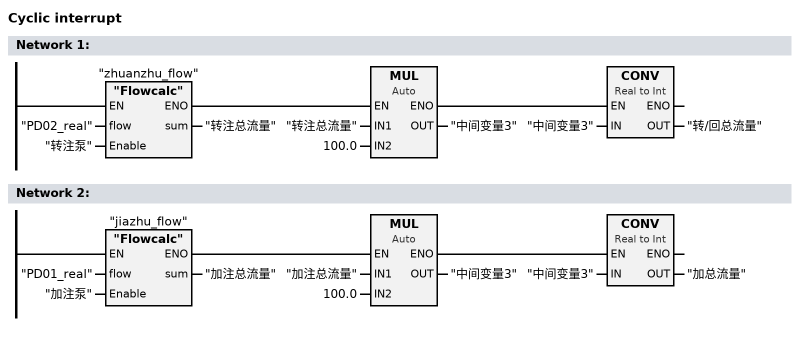
   RUNG wire#powerrail
      "zhuanzhu_flow"(flow := "PD02_real", Enable := "转注泵", sum => "转注总流量")
      { S7_GenerateENO := "TRUE" } Mul(in1 := "转注总流量", in2 := 100.0, out => "中间变量3")
      { S7_Templates := "[SrcType := Real, DestType := Int]"; S7_GenerateENO := "TRUE" } Convert(in := "中间变量3", out => "转/回总流量")
   END_RUNG
   // the same network as SCL:
   // ENO of a box is taken as its EN; it also drops when the box reports an error
   "zhuanzhu_flow"(flow := "PD02_real", Enable := "转注泵", sum => "转注总流量", ENO => #_w1);   // "Flowcalc"
   IF #_w1 THEN
       "中间变量3" := "转注总流量" * 100.0;
       "转/回总流量" := REAL_TO_INT("中间变量3");
   END_IF;
END_REGION

REGION Network 2
   RUNG wire#powerrail
      "jiazhu_flow"(flow := "PD01_real", Enable := "加注泵", sum => "加注总流量")
      { S7_GenerateENO := "TRUE" } Mul(in1 := "加注总流量", in2 := 100.0, out => "中间变量3")
      { S7_Templates := "[SrcType := Real, DestType := Int]"; S7_GenerateENO := "TRUE" } Convert(in := "中间变量3", out => "加总流量")
   END_RUNG
   // the same network as SCL:
   // ENO of a box is taken as its EN; it also drops when the box reports an error
   "jiazhu_flow"(flow := "PD01_real", Enable := "加注泵", sum => "加注总流量", ENO => #_w1);   // "Flowcalc"
   IF #_w1 THEN
       "中间变量3" := "加注总流量" * 100.0;
       "加总流量" := REAL_TO_INT("中间变量3");
   END_IF;
END_REGION
END_ORGANIZATION_BLOCK